Fanuc KAREL source: kb00193.KL

-- PROVISIONAL review KL for V770-1; original PC SHA256 b72202b071c8caad40a6155ef845a404e76afddf977e04f406f807c1271c1e78
-- Incomplete behavior may be omitted. Consult companion uncertainty JSON. Do not deploy.
PROGRAM KB00193
%NOLOCKGROUP
BEGIN
  -- UNRESOLVED_PC offsets 5-12; opcodes 9D,23
  -- UNRESOLVED_PC offsets 17-24; opcodes 9D,23
  -- UNRESOLVED_PC offsets 29-45; opcodes 27,22,22,31
  -- UNRESOLVED_PC offsets 50-54; opcodes 7F
END KB00193
